Fanuc KAREL source: kf00098.KL

-- PROVISIONAL review KL for V940-1; original PC SHA256 3e651a630b2e94eb7f80599199318565e0fe020e813d3d9091d7727710e40e99
-- Incomplete behavior may be omitted. Consult companion uncertainty JSON. Do not deploy.
PROGRAM KF00098
%NOLOCKGROUP
BEGIN
  -- V9_ZERO_TABLE_METADATA_HINT layout=0002_ascii; no indexed target words; source/name/runtime held
  -- UNRESOLVED_PC offsets 5-16; opcodes 2E,23
  -- UNRESOLVED_PC offsets 21-32; opcodes 2E,23
  -- UNRESOLVED_PC offsets 37-55; opcodes 27,27,9D,22,22,31
  -- UNRESOLVED_PC offsets 60-64; opcodes 7F
END KF00098
